(* PLC project  *)

CONFIGURATION EtherCAT
END_CONFIGURATION
